// TIA Portal V19 export
DATA_BLOCK "PPrgArchive17"   // DB512
// stored: IsOnlyStoredInLoadMemory true, MemoryReserve 0, Namespace G
   VAR RETAIN
      PRG : Array[1601..1700] of "PPrg_Data";
   END_VAR
BEGIN
END_DATA_BLOCK
